// TIA Portal V19 export
DATA_BLOCK "CallEquipment_DB"   // DB64
AUTHOR : Siemens_FA_SUP
// stored: InstanceOfName Unit3.EM1.CallEquipment, InstanceOfType FB, Namespace Unit3.EM1
"Unit3.EM1.CallEquipment"
   // VAR_IN_OUT
   //    unitStatus : "LAF_typeUnitStatus";
   //    unitAlarmDB : "LAF_typeAlarms";
   //    emFeedback : "LUC_typeEmFeedback";
   // END_VAR
   // VAR
   //    statUnitStatus { ExternalWritable := 'False'} : "LAF_typeUnitStatus";
   //    instSequence { ExternalWritable := 'False'} : "Unit3.EM1.Sequence";
   //    instManageBitAlarms { ExternalWritable := 'False'} : "LAF_ManageBitAlarms";
   //    instHoldingJob { ExternalWritable := 'False'; S7_SetPoint := 'True'} : "LAF_SelectJob";
   //    instUnholdingJob { ExternalWritable := 'False'; S7_SetPoint := 'True'} : "LAF_SelectJob";
   //    instStartingJob { ExternalWritable := 'False'} : "LAF_SelectJob";
   //    instPosMovingJob { ExternalWritable := 'False'; S7_SetPoint := 'True'} : "LAF_SelectJob";
   //    instStoppingJob { ExternalWritable := 'False'; S7_SetPoint := 'True'} : "LAF_SelectJob";
   //    instHomeJob { ExternalWritable := 'False'; S7_SetPoint := 'True'} : "LAF_SelectJob";
   //    instResetingJob { ExternalWritable := 'False'; S7_SetPoint := 'True'} : "LAF_SelectJob";
   //    instSpecialFuncAbsPos { ExternalWritable := 'False'; S7_SetPoint := 'True'} : "LAF_SelectJob";
   //    instCm2AxisPos { ExternalWritable := 'False'; S7_SetPoint := 'True'} : "LBC_AxisSimpleControl";
   //    instCmReset { ExternalWritable := 'False'; S7_SetPoint := 'True'} : "Unit3.EM1.EXCHANGETRAY_CmResetOperator";
   //    instCm1SingleTm { ExternalWritable := 'False'; S7_SetPoint := 'True'} : "LEXCHANGETRAY_U3Em1SingleTM";
   //    instCm3NgStrap { ExternalWritable := 'False'; S7_SetPoint := 'True'} : "LEXCHANGETRAY_NgStrapDetect";
   //    instCm4FrButton { ExternalWritable := 'False'; S7_SetPoint := 'True'} : "LEXCHANGETRAY_FrButtonTm";
   //    statHomingJobStartCondition { ExternalWritable := 'False'; S7_SetPoint := 'True'} : Bool;
   //    statPosMovingJobStartCondition { ExternalWritable := 'False'} : Bool;
   //    statLstUnitMode { ExternalWritable := 'False'; S7_SetPoint := 'True'} : DInt;
   //    statLstUnitStatus { ExternalWritable := 'False'} : DInt;
   //    statLstCurrentStep { ExternalWritable := 'False'} : DInt;
   //    statJobComplete { ExternalWritable := 'False'} : Bool;
   // END_VAR
BEGIN
END_DATA_BLOCK
